(* CODESYS project twincat_implementation.library
   TcLibraryId: TE140x Module Vendor|twincat_implementation|0.0.0.1
   Company: TE140x Module Vendor
   DefaultNamespace: twincat_implementation
   Version: 0.0.0.1
   Placeholder: twincat_implementation
   Title: twincat_implementation

Project tree, tasks and I/O mapping:
  Version/
    global variables Global_Version
  POUs/
    function block FB_twincat_implementation [ST]: FB_exit, FB_init, nHResult, eInitExceptionHandling, eUpdateExceptionHandling, nExceptionCnt, stActiveException, bInitialized, bExecute
  DUTs/
    data type ST_FB_twincat_implementation_FB_Main
    data type ST_FB_twincat_implementation_FB_exit
    data type ST_FB_twincat_implementation_FB_init
    data type ST_GetSet_HRESULT
    data type E_FpExcptCtrlSetEx
    data type ST_GetSet_E_FpExcptCtrlSetEx
    data type ST_GetSet_ULINT
    data type ST_ExceptionInfo
    data type ST_GetSet_ST_ExceptionInfo
    data type ST_GetSet_BOOL
    data type T_matrix_2_real_T
    data type T_matrix_4_real_T
    data type ST_B_twincat_implementation_T
    data type T_int_T
    data type ST_DW_twincat_implementation_T
    data type ST_ExtU_twincat_implementation_T
    data type ST_ExtY_twincat_implementation_T
    data type ST_P_twincat_implementation_T
    data type T_matrix_2_boolean_T
    data type ST_XDis_twincat_implementation_T
    data type ST_X_twincat_implementation_T
*)

// DUTs/ST_FB_twincat_implementation_FB_Main

	{attribute 'TcIecLibraryType'}
{attribute 'hide'}
TYPE ST_FB_twincat_implementation_FB_Main : 
	STRUCT
		 {attribute 'GUID' := '18071995-0000-0000-0000-000000000018'}
		pInst : PVOID;
		result : BOOL;
		 {attribute 'hide'}
		_reserved1 : UINT_24_56;
	END_STRUCT
END_TYPE

// DUTs/ST_FB_twincat_implementation_FB_exit

	{attribute 'TcIecLibraryType'}
{attribute 'hide'}
TYPE ST_FB_twincat_implementation_FB_exit : 
	STRUCT
		 {attribute 'GUID' := '18071995-0000-0000-0000-000000000018'}
		pInst : PVOID;
		bInCopyCode : BOOL;
		result : BOOL;
		 {attribute 'hide'}
		_reserved1 : UINT_16_48;
	END_STRUCT
END_TYPE

// DUTs/ST_FB_twincat_implementation_FB_init

	{attribute 'TcIecLibraryType'}
{attribute 'hide'}
TYPE ST_FB_twincat_implementation_FB_init : 
	STRUCT
		 {attribute 'GUID' := '18071995-0000-0000-0000-000000000018'}
		pInst : PVOID;
		bInitRetains : BOOL;
		bInCopyCode : BOOL;
		result : BOOL;
		 {attribute 'hide'}
		_reserved1 : UINT_8_40;
	END_STRUCT
END_TYPE

// DUTs/ST_GetSet_HRESULT

	{attribute 'TcIecLibraryType'}
{attribute 'hide'}
TYPE ST_GetSet_HRESULT : 
	STRUCT
		 {attribute 'GUID' := '18071995-0000-0000-0000-000000000018'}
		pInst : PVOID;
		 {attribute 'GUID' := '18071995-0000-0000-0000-000000000019'}
		nParam : HRESULT;
		 {attribute 'hide'}
		_reserved1 : UINT_0_32;
	END_STRUCT
END_TYPE

// DUTs/E_FpExcptCtrlSetEx

(* Generated from type 'TcMgSdk.FpExcptCtrlSetEx' *)
	{attribute 'TcIecLibraryType'}
TYPE E_FpExcptCtrlSetEx : (
	CallerExceptions:=1, 	(* Use the floating point exception settings provided by the caller *)
	ThrowExceptions:=3, 	(* Enable floating point exceptions on invalid operations and divisions by zero *)
	SuppressExceptions:=13, 	(* Disable floating point exceptions. *)
	LogExceptions:=19, 	(* Log exception information. *)
	LogAndHold:=51, 	(* Log exception information and puase execution of the cyclic code after completion of the actual cycle *)
	LogAndCatch:=83, 	(* Log exception information and immediately terminate execution of the cyclic code. Reinitialization is required to restart. *)
	LogAndDump:=147, 	(* Log exception information, create a dump file with detailed exception information and try to continue execution of the cyclic code *)
	LogHoldAndDump:=179, 	(* Log exception information, create a dump file with detailed exception information and puase execution of the cyclic code after completion of the actual cycle *)
	LogCatchAndDump:=211	(* Log exception information, create a dump file with detailed exception information and immediately terminate execution of the cyclic code. Reinitialization is required to restart. *)
) USINT;
END_TYPE

// DUTs/ST_GetSet_E_FpExcptCtrlSetEx

	{attribute 'TcIecLibraryType'}
{attribute 'hide'}
TYPE ST_GetSet_E_FpExcptCtrlSetEx : 
	STRUCT
		 {attribute 'GUID' := '18071995-0000-0000-0000-000000000018'}
		pInst : PVOID;
		eParam : E_FpExcptCtrlSetEx;
		 {attribute 'hide'}
		_reserved1 : UINT_24_56;
	END_STRUCT
END_TYPE

// DUTs/ST_GetSet_ULINT

	{attribute 'TcIecLibraryType'}
{attribute 'hide'}
TYPE ST_GetSet_ULINT : 
	STRUCT
		 {attribute 'GUID' := '18071995-0000-0000-0000-000000000018'}
		pInst : PVOID;
		nParam : ULINT;
	END_STRUCT
END_TYPE

// DUTs/ST_ExceptionInfo

(* Generated from type 'TcMgSdk.ExceptionInfo' *)
	{attribute 'TcIecLibraryType'}
TYPE ST_ExceptionInfo : 
	STRUCT
		(* Generated from item 'ExceptionCode' *)
		nExceptionCode : DINT;
		(* Generated from item 'TmxName' *)
		 {attribute 'GUID' := '18071995-0000-0000-0000-00010000007F'}
		sTmxName : STRING(127);
		(* Generated from item 'TmxVersion' *)
		nTmxVersion : ARRAY [0..3] OF UDINT;
		(* Generated from item 'InstructionAddr' *)
		nInstructionAddr : UDINT;
		(* Generated from item 'ReturnAddr' *)
		nReturnAddr : ARRAY [0..3] OF UDINT;
		(* Generated from item 'DumpCreated' *)
		bDumpCreated : BOOL;
		 {attribute 'hide'}
		_reserved1 : ARRAY [1..3] OF USINT;
	END_STRUCT
END_TYPE

// DUTs/ST_GetSet_ST_ExceptionInfo

	{attribute 'TcIecLibraryType'}
{attribute 'hide'}
TYPE ST_GetSet_ST_ExceptionInfo : 
	STRUCT
		 {attribute 'GUID' := '18071995-0000-0000-0000-000000000018'}
		pInst : PVOID;
		stParam : ST_ExceptionInfo;
		 {attribute 'hide'}
		_reserved1 : UINT_0_32;
	END_STRUCT
END_TYPE

// DUTs/ST_GetSet_BOOL

	{attribute 'TcIecLibraryType'}
{attribute 'hide'}
TYPE ST_GetSet_BOOL : 
	STRUCT
		 {attribute 'GUID' := '18071995-0000-0000-0000-000000000018'}
		pInst : PVOID;
		bParam : BOOL;
		 {attribute 'hide'}
		_reserved1 : UINT_24_56;
	END_STRUCT
END_TYPE

// DUTs/T_matrix_2_real_T

(* Generated from type 'matrix_2_real_T' *)
	{attribute 'TcIecLibraryType'}
TYPE T_matrix_2_real_T : ARRAY [0..1] OF LREAL;
END_TYPE

// DUTs/T_matrix_4_real_T

(* Generated from type 'matrix_4_real_T' *)
	{attribute 'TcIecLibraryType'}
TYPE T_matrix_4_real_T : ARRAY [0..3] OF LREAL;
END_TYPE

// DUTs/ST_B_twincat_implementation_T

(* Generated from type 'B_twincat_implementation_T' *)
	{attribute 'TcIecLibraryType'}
TYPE ST_B_twincat_implementation_T : 
	STRUCT
		(* Generated from item 'X0' *)
		aX0 : T_matrix_2_real_T;
		(* Generated from item 'MemoryX' *)
		aMemoryX : T_matrix_2_real_T;
		(* Generated from item 'Sum' *)
		fSum : LREAL;
		(* Generated from item 'Add' *)
		aAdd : T_matrix_2_real_T;
		(* Generated from item 'Product3' *)
		aProduct3 : T_matrix_2_real_T;
		(* Generated from item 'P' *)
		aP : T_matrix_4_real_T;
		(* Generated from item 'Akxhatkk1' *)
		aAkxhatkk1 : T_matrix_2_real_T;
		(* Generated from item 'Bkuk' *)
		aBkuk : T_matrix_2_real_T;
		(* Generated from item 'Dkuk' *)
		fDkuk : LREAL;
		(* Generated from item 'Sum_p' *)
		fSum_p : LREAL;
	END_STRUCT
END_TYPE

// DUTs/T_int_T

(* Generated from type 'int_T' *)
	{attribute 'TcIecLibraryType'}
TYPE T_int_T : DINT;
END_TYPE

// DUTs/ST_DW_twincat_implementation_T

(* Generated from type 'DW_twincat_implementation_T' *)
	{attribute 'TcIecLibraryType'}
TYPE ST_DW_twincat_implementation_T : 
	STRUCT
		(* Generated from item 'MemoryX_IWORK' *)
		nMemoryX_IWORK : T_int_T;
		(* Generated from item 'MeasurementUpdate_MODE' *)
		bMeasurementUpdate_MODE : BOOL;
		 {attribute 'hide'}
		_reserved1 : ARRAY [1..3] OF USINT;
	END_STRUCT
END_TYPE

// DUTs/ST_ExtU_twincat_implementation_T

(* Generated from type 'ExtU_twincat_implementation_T' *)
	{attribute 'TcIecLibraryType'}
TYPE ST_ExtU_twincat_implementation_T : 
	STRUCT
		(* Generated from item 'ddx_f' *)
		fddx_f : LREAL;
	END_STRUCT
END_TYPE

// DUTs/ST_ExtY_twincat_implementation_T

(* Generated from type 'ExtY_twincat_implementation_T' *)
	{attribute 'TcIecLibraryType'}
TYPE ST_ExtY_twincat_implementation_T : 
	STRUCT
		(* Generated from item 'torque' *)
		ftorque : LREAL;
	END_STRUCT
END_TYPE

// DUTs/ST_P_twincat_implementation_T

(* Generated from type 'P_twincat_implementation_T' *)
	{attribute 'TcIecLibraryType'}
TYPE ST_P_twincat_implementation_T : 
	STRUCT
		(* Generated from item 'K' *)
		aK : T_matrix_2_real_T;
		(* Generated from item 'Lykyhatkk1_Y0' *)
		fLykyhatkk1_Y0 : LREAL;
		(* Generated from item 'Constant_Value' *)
		fConstant_Value : LREAL;
		(* Generated from item 'X0_Value' *)
		aX0_Value : T_matrix_2_real_T;
		(* Generated from item 'Saturation_UpperSat' *)
		fSaturation_UpperSat : LREAL;
		(* Generated from item 'Saturation_LowerSat' *)
		fSaturation_LowerSat : LREAL;
		(* Generated from item 'A_Value' *)
		aA_Value : T_matrix_4_real_T;
		(* Generated from item 'B_Value' *)
		aB_Value : T_matrix_2_real_T;
		(* Generated from item 'C_Value' *)
		aC_Value : T_matrix_2_real_T;
		(* Generated from item 'CovarianceZ_Value' *)
		aCovarianceZ_Value : T_matrix_4_real_T;
		(* Generated from item 'KalmanGainL_Value' *)
		aKalmanGainL_Value : T_matrix_2_real_T;
		(* Generated from item 'D_Value' *)
		fD_Value : LREAL;
		(* Generated from item 'isSqrtUsed_Value' *)
		bisSqrtUsed_Value : BOOL;
		(* Generated from item 'Enable_Value' *)
		bEnable_Value : BOOL;
		 {attribute 'hide'}
		_reserved1 : ARRAY [1..6] OF USINT;
	END_STRUCT
END_TYPE

// DUTs/T_matrix_2_boolean_T

(* Generated from type 'matrix_2_boolean_T' *)
	{attribute 'TcIecLibraryType'}
{attribute 'BaseTypeGUID' := '18071995-0000-0000-0000-000000000030'}
TYPE T_matrix_2_boolean_T : ARRAY [0..1] OF BOOL;
END_TYPE

// DUTs/ST_XDis_twincat_implementation_T

(* Generated from type 'XDis_twincat_implementation_T' *)
	{attribute 'TcIecLibraryType'}
TYPE ST_XDis_twincat_implementation_T : 
	STRUCT
		(* Generated from item 'MemoryX_CSTATE' *)
		aMemoryX_CSTATE : T_matrix_2_boolean_T;
	END_STRUCT
END_TYPE

// DUTs/ST_X_twincat_implementation_T

(* Generated from type 'X_twincat_implementation_T' *)
	{attribute 'TcIecLibraryType'}
TYPE ST_X_twincat_implementation_T : 
	STRUCT
		(* Generated from item 'MemoryX_CSTATE' *)
		aMemoryX_CSTATE : T_matrix_2_real_T;
	END_STRUCT
END_TYPE

// Version/Global_Version
{attribute 'TcGenerated'}
// This function has been automatically generated from the project information.
VAR_GLOBAL CONSTANT
	{attribute 'const_non_replaced'}
	{attribute 'linkalways'}
	stLibVersion_twincat_implementation : ST_LibVersion := (iMajor := 0, iMinor := 0, iBuild := 0, iRevision := 1, sVersion := '0.0.0.1');
	{attribute 'const_non_replaced'}
	{attribute 'linkalways'}
	sLibraryId_twincat_implementation : String := 'TE140x Module Vendor|twincat_implementation|0.0.0.1';
END_VAR

// POUs/FB_twincat_implementation

	{attribute 'c++_compatible'}
	{attribute 'external_name' := 'FB_twincat_implementation_GUID_94B38E83_2E40_E9F5_2B21_7D947837890F'}
	{attribute 'TcIecLibraryType'}
	{attribute 'reflection'}
	FUNCTION_BLOCK FB_twincat_implementation
	VAR
		{attribute 'hide'}
		{attribute 'no_copy'}
		 {attribute 'GUID' := '18071995-0000-0000-0000-000000000018'}
		m_pData : PVOID;
		{attribute 'TcInitSymbol'}
		 {attribute 'GUID' := '8007AE3B-86BB-40F2-B385-EF87FCC239A4'}
		eTraceLevelMax : TcTraceLevel := TcTraceLevel.tlInfo;
		 {attribute 'hide'}
		_reserved1 : UDINT;
		{attribute 'hide'}
		{attribute 'instance-path'}
		{attribute 'noinit'}
		 {attribute 'GUID' := '18071995-0000-0000-0000-0001000000FF'}
		sInstancePath : STRING(255);
		{attribute 'hide'}
		{attribute 'noinit'}
		 {attribute 'GUID' := '18071995-0000-0000-0000-000000000019'}
		m_HResultLog : HRESULT;
		{attribute 'hide'}
		{attribute 'noinit'}
		 {attribute 'GUID' := '18071995-0000-0000-0000-000000000019'}
		m_HResult : HRESULT;
		 {attribute 'hide'}
		_reserved2 : ARRAY [1..184] OF USINT;
		{attribute 'hide'}
		{attribute 'no_copy'}
		m_ExtModeData : ULINT;
	END_VAR
	VAR_INPUT
		(* Generated from item 'ddx_f' *)
		fddx_f : LREAL;
	END_VAR
	VAR_OUTPUT
		(* Generated from item 'torque' *)
		ftorque : LREAL;
	END_VAR
	VAR
		(* Generated from item 'Ptwincat_implementation_M' *)
		 {attribute 'GUID' := '18071995-0000-0000-0000-000000000018'}
		pPtwincat_implementation_M : PVOID;
	END_VAR


	METHOD FB_exit : BOOL
	VAR_INPUT
		bInCopyCode : BOOL;
	END_VAR
END_METHOD


	METHOD FB_init : BOOL
	VAR_INPUT
		bInitRetains : BOOL;
		bInCopyCode : BOOL;
	END_VAR
END_METHOD


{attribute 'monitoring' := 'call'}
	PROPERTY nHResult : HRESULT
GET
END_GET
END_PROPERTY


{attribute 'monitoring' := 'call'}
	PROPERTY eInitExceptionHandling : E_FpExcptCtrlSetEx
GET
END_GET
SET
END_SET
END_PROPERTY


{attribute 'monitoring' := 'call'}
	PROPERTY eUpdateExceptionHandling : E_FpExcptCtrlSetEx
GET
END_GET
SET
END_SET
END_PROPERTY


{attribute 'monitoring' := 'call'}
	PROPERTY nExceptionCnt : ULINT
GET
END_GET
END_PROPERTY


{attribute 'monitoring' := 'variable'}
	PROPERTY stActiveException : ST_ExceptionInfo
GET
END_GET
END_PROPERTY


{attribute 'monitoring' := 'call'}
	PROPERTY bInitialized : BOOL
GET
END_GET
END_PROPERTY


{attribute 'monitoring' := 'call'}
	PROPERTY bExecute : BOOL
GET
END_GET
SET
END_SET
END_PROPERTY

END_FUNCTION_BLOCK
